// TIA Portal V20 export
FUNCTION "CallDiagnostic" : Void   // FC16, LAD
TITLE = Diagnose / Diagnostics
AUTHOR : SICAR
FAMILY : Diag
// Aufruf: Diagnose / Call of SICAR Diagnostic blocks
// stored: IsIECCheckEnabled true, SetENOAutomatically true
   VAR_TEMP
      statWStringName : WString[24];
      tempHardwareOKexample : Bool;   // REPLACE: This output can be used as an interlock for Control Modules
   END_VAR
   // Ret_Val : Ret_Val
   VAR_TEMP   // added for the SCL form of the ladder/FBD networks
      _w1 : Bool;
   END_VAR
BEGIN

REGION Network 1: Beschreibung / BLOCK INFO HEADER
   // **Betriebsart Automatik / Hand**  
   // Der Baustein ist keiner Betriebsart / Betriebsartenbereich zugeordnet.  
   // 
   // **Alarme**  
   // Der Baustein generiert keine Alarme.  
   // 
   // #### PLC-Datentypen  
   // Verwendete PLC-Datentypen für den SPS-Programmbaustein und das zugehörige WinCC-Bild.  
   // 
   // {.pageWidth}
   // ![Image](CallInterfaceSignals/de/image1.PNG)
   //  
   //  
   // #### Bausteinaufrufe 
   // Der Baustein “LSicar_InterfaceSignalsBool“ wird in diesem FB als Multi-Instanz aufgerufen, entspr. nebenstehender beispielhafter Darstellung.  
   // 
   // {.pageWidth}
   // ![Image](CallInterfaceSignals/de/image2.PNG)
   //  
   // Um einen neuen FB aufzurufen, ziehen Sie den FB in ein neues Netzwerk, wählen Sie „Multiinstanz“ aus, vergeben Sie einen Namen und parametrieren Sie den FB-Aufruf.  
   // 
   // {.pageWidth}
   // ![Image](CallInterfaceSignals/de/image3.PNG)
   //  
   //  
   // #### Weitere Hinweise 
   // 
   // #### Updateinfo 
   // 
   // #### Weitere Dokumente 
   // 
   // ![Icon](_Icon/reference.PNG)
   // 
   // ..\Library Types\LSicar_InterfaceSignalsBool.pdf
   // SIEMENS AG / (c)Copyright 2023
   // ------------------------------------------------------------------------------
   // Title:            CallDiagnostic (FC16)
   // Comment/Function: Call of SICAR Diagnostic blocks
   // Library/Family:   Diag
   // Author:           SICAR
   // Tested with:      ---
   // Engineering:      TIA Portal V19
   // Restrictions:     -
   // Requirements:     ---
   // ------------------------------------------------------------------------------
   // Change log table:
   // Version | Date | Expert in charge | Changes applied
   // -------|---------|-------------|--------------------------------------------
   // 01.00.00 | 01.01.1999 | Person x | First released version
   // 01.00.01 | 02.01.1999 | Person y | Block was Updated
END_REGION

REGION Network 2: Call: Diagnostic Profinet Devices
   // For diagnose the whole profinet devices of this PLC
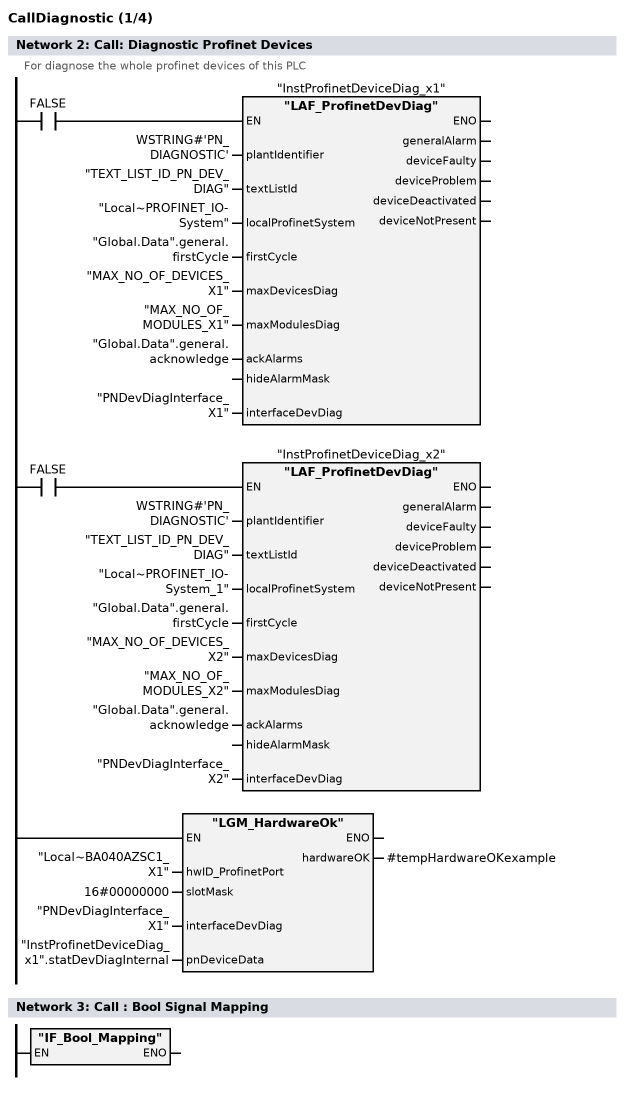
   RUNG wire#powerrail
      Contact( FALSE )
      "InstProfinetDeviceDiag_x1"(plantIdentifier := WSTRING#'PN_DIAGNOSTIC', textListId := "TEXT_LIST_ID_PN_DEV_DIAG", localProfinetSystem := "Local~PROFINET_IO-System", firstCycle := "Global.Data".general.firstCycle, maxDevicesDiag := "MAX_NO_OF_DEVICES_X1", maxModulesDiag := "MAX_NO_OF_MODULES_X1", ackAlarms := "Global.Data".general.acknowledge, hideAlarmMask :=, interfaceDevDiag := "PNDevDiagInterface_X1", generalAlarm =>, deviceFaulty =>, deviceProblem =>, deviceDeactivated =>, deviceNotPresent =>)
   END_RUNG
   RUNG wire#powerrail
      Contact( FALSE )
      "InstProfinetDeviceDiag_x2"(plantIdentifier := WSTRING#'PN_DIAGNOSTIC', textListId := "TEXT_LIST_ID_PN_DEV_DIAG", localProfinetSystem := "Local~PROFINET_IO-System_1", firstCycle := "Global.Data".general.firstCycle, maxDevicesDiag := "MAX_NO_OF_DEVICES_X2", maxModulesDiag := "MAX_NO_OF_MODULES_X2", ackAlarms := "Global.Data".general.acknowledge, hideAlarmMask :=, interfaceDevDiag := "PNDevDiagInterface_X2", generalAlarm =>, deviceFaulty =>, deviceProblem =>, deviceDeactivated =>, deviceNotPresent =>)
   END_RUNG
   RUNG wire#powerrail
      "LGM_HardwareOk"(hwID_ProfinetPort := "Local~BA040AZSC1_X1", slotMask := 16#00000000, interfaceDevDiag := "PNDevDiagInterface_X1", pnDeviceData := "InstProfinetDeviceDiag_x1".statDevDiagInternal, hardwareOK => #tempHardwareOKexample)
   END_RUNG
   // the same network as SCL:
   IF FALSE THEN
       "InstProfinetDeviceDiag_x1"(plantIdentifier := WSTRING#'PN_DIAGNOSTIC',   // "LAF_ProfinetDevDiag"
                               textListId := "TEXT_LIST_ID_PN_DEV_DIAG",
                               localProfinetSystem := "Local~PROFINET_IO-System",
                               firstCycle := "Global.Data".general.firstCycle,
                               maxDevicesDiag := "MAX_NO_OF_DEVICES_X1",
                               maxModulesDiag := "MAX_NO_OF_MODULES_X1",
                               ackAlarms := "Global.Data".general.acknowledge,
                               interfaceDevDiag := "PNDevDiagInterface_X1");
       "InstProfinetDeviceDiag_x2"(plantIdentifier := WSTRING#'PN_DIAGNOSTIC',   // "LAF_ProfinetDevDiag"
                               textListId := "TEXT_LIST_ID_PN_DEV_DIAG",
                               localProfinetSystem := "Local~PROFINET_IO-System_1",
                               firstCycle := "Global.Data".general.firstCycle,
                               maxDevicesDiag := "MAX_NO_OF_DEVICES_X2",
                               maxModulesDiag := "MAX_NO_OF_MODULES_X2",
                               ackAlarms := "Global.Data".general.acknowledge,
                               interfaceDevDiag := "PNDevDiagInterface_X2");
   END_IF;
   "LGM_HardwareOk"(hwID_ProfinetPort := "Local~BA040AZSC1_X1",
                    slotMask := 16#00000000,
                    interfaceDevDiag := "PNDevDiagInterface_X1",
                    pnDeviceData := "InstProfinetDeviceDiag_x1".statDevDiagInternal,
                    hardwareOK => #tempHardwareOKexample);
END_REGION

REGION Network 3: Call : Bool Signal Mapping
   RUNG wire#powerrail
      "IF_Bool_Mapping"()
   END_RUNG
   // the same network as SCL:
   "IF_Bool_Mapping"();
END_REGION

REGION Network 4: Call: Diagnostic Bool Interface Signals
   // Call the interface bool blocks to show boolean signals on the HMI
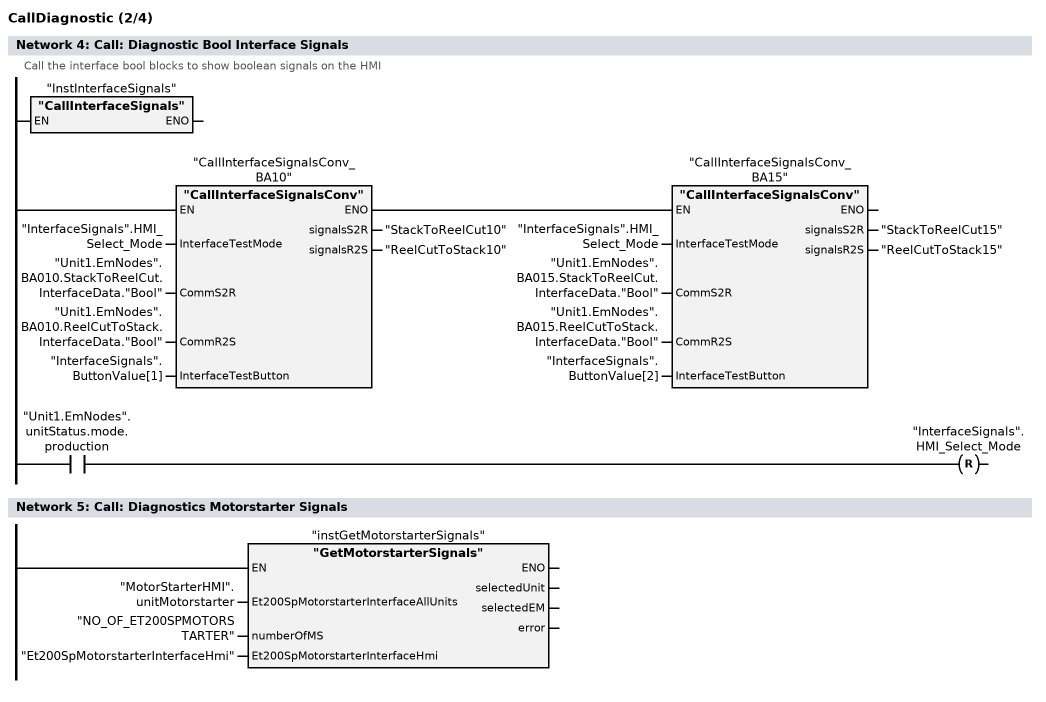
   RUNG wire#powerrail
      "InstInterfaceSignals"()
   END_RUNG
   RUNG wire#powerrail
      "CallInterfaceSignalsConv_BA10"(InterfaceTestMode := "InterfaceSignals".HMI_Select_Mode, CommS2R := "Unit1.EmNodes".BA010.StackToReelCut.InterfaceData."Bool", CommR2S := "Unit1.EmNodes".BA010.ReelCutToStack.InterfaceData."Bool", InterfaceTestButton := "InterfaceSignals".ButtonValue[1], signalsS2R => "StackToReelCut10", signalsR2S => "ReelCutToStack10")
      "CallInterfaceSignalsConv_BA15"(InterfaceTestMode := "InterfaceSignals".HMI_Select_Mode, CommS2R := "Unit1.EmNodes".BA015.StackToReelCut.InterfaceData."Bool", CommR2S := "Unit1.EmNodes".BA015.ReelCutToStack.InterfaceData."Bool", InterfaceTestButton := "InterfaceSignals".ButtonValue[2], signalsS2R => "StackToReelCut15", signalsR2S => "ReelCutToStack15")
   END_RUNG
   RUNG wire#powerrail
      Contact( "Unit1.EmNodes".unitStatus.mode.production )
      R_Coil( "InterfaceSignals".HMI_Select_Mode )
   END_RUNG
   // the same network as SCL:
   "InstInterfaceSignals"();   // "CallInterfaceSignals"
   "CallInterfaceSignalsConv_BA10"(InterfaceTestMode := "InterfaceSignals".HMI_Select_Mode,   // "CallInterfaceSignalsConv"
                           CommS2R := "Unit1.EmNodes".BA010.StackToReelCut.InterfaceData."Bool",
                           CommR2S := "Unit1.EmNodes".BA010.ReelCutToStack.InterfaceData."Bool",
                           InterfaceTestButton := "InterfaceSignals".ButtonValue[1],
                           signalsS2R => "StackToReelCut10",
                           signalsR2S => "ReelCutToStack10",
                           ENO => #_w1);
   IF #_w1 THEN
       "CallInterfaceSignalsConv_BA15"(InterfaceTestMode := "InterfaceSignals".HMI_Select_Mode,   // "CallInterfaceSignalsConv"
                               CommS2R := "Unit1.EmNodes".BA015.StackToReelCut.InterfaceData."Bool",
                               CommR2S := "Unit1.EmNodes".BA015.ReelCutToStack.InterfaceData."Bool",
                               InterfaceTestButton := "InterfaceSignals".ButtonValue[2],
                               signalsS2R => "StackToReelCut15",
                               signalsR2S => "ReelCutToStack15");
   END_IF;
   IF "Unit1.EmNodes".unitStatus.mode.production THEN "InterfaceSignals".HMI_Select_Mode := FALSE; END_IF;
END_REGION

REGION Network 5: Call: Diagnostics Motorstarter Signals
   RUNG wire#powerrail
      "instGetMotorstarterSignals"(Et200SpMotorstarterInterfaceAllUnits := "MotorStarterHMI".unitMotorstarter, numberOfMS := "NO_OF_ET200SPMOTORSTARTER", Et200SpMotorstarterInterfaceHmi := "Et200SpMotorstarterInterfaceHmi", selectedUnit =>, selectedEM =>, error =>)
   END_RUNG
   // the same network as SCL:
   "instGetMotorstarterSignals"(Et200SpMotorstarterInterfaceAllUnits := "MotorStarterHMI".unitMotorstarter,   // "GetMotorstarterSignals"
                           numberOfMS := "NO_OF_ET200SPMOTORSTARTER",
                           Et200SpMotorstarterInterfaceHmi := "Et200SpMotorstarterInterfaceHmi");
END_REGION

REGION Network 6: Call: Diagnostics Drives
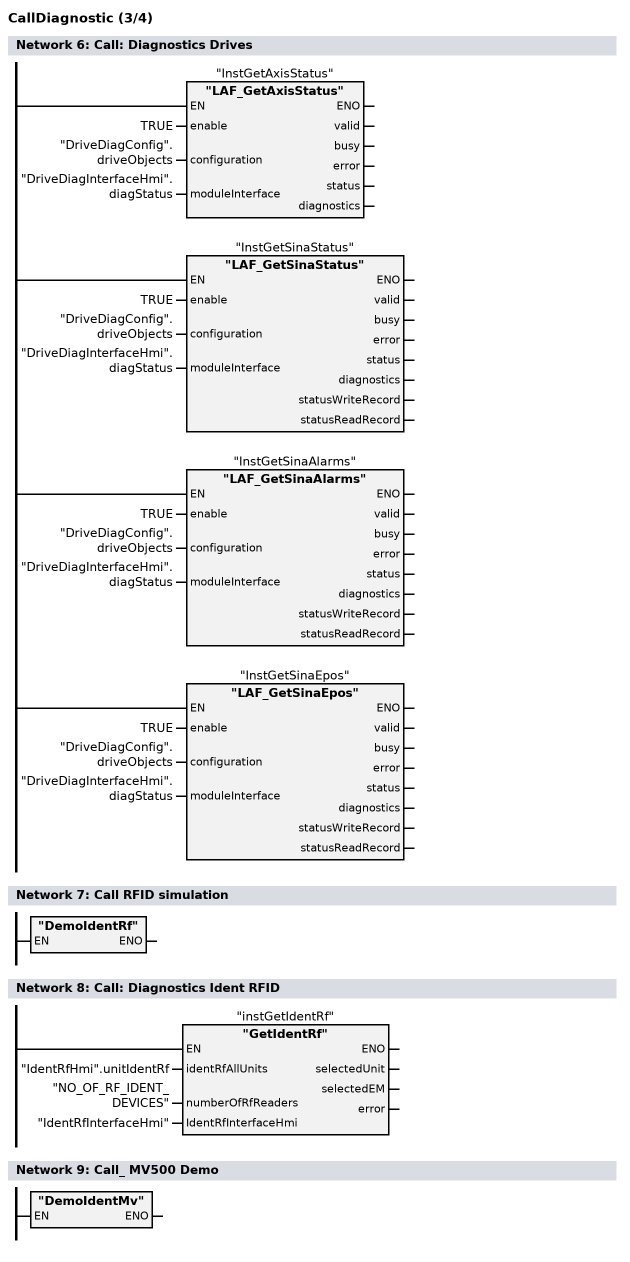
   RUNG wire#powerrail
      "InstGetAxisStatus"(enable := TRUE, configuration := "DriveDiagConfig".driveObjects, moduleInterface := "DriveDiagInterfaceHmi".diagStatus, valid =>, busy =>, error =>, status =>, diagnostics =>)
   END_RUNG
   RUNG wire#powerrail
      "InstGetSinaStatus"(enable := TRUE, configuration := "DriveDiagConfig".driveObjects, moduleInterface := "DriveDiagInterfaceHmi".diagStatus, valid =>, busy =>, error =>, status =>, diagnostics =>, statusWriteRecord =>, statusReadRecord =>)
   END_RUNG
   RUNG wire#powerrail
      "InstGetSinaAlarms"(enable := TRUE, configuration := "DriveDiagConfig".driveObjects, moduleInterface := "DriveDiagInterfaceHmi".diagStatus, valid =>, busy =>, error =>, status =>, diagnostics =>, statusWriteRecord =>, statusReadRecord =>)
   END_RUNG
   RUNG wire#powerrail
      "InstGetSinaEpos"(enable := TRUE, configuration := "DriveDiagConfig".driveObjects, moduleInterface := "DriveDiagInterfaceHmi".diagStatus, valid =>, busy =>, error =>, status =>, diagnostics =>, statusWriteRecord =>, statusReadRecord =>)
   END_RUNG
   // the same network as SCL:
   "InstGetAxisStatus"(enable := TRUE,   // "LAF_GetAxisStatus"
                       configuration := "DriveDiagConfig".driveObjects,
                       moduleInterface := "DriveDiagInterfaceHmi".diagStatus);
   "InstGetSinaStatus"(enable := TRUE,   // "LAF_GetSinaStatus"
                       configuration := "DriveDiagConfig".driveObjects,
                       moduleInterface := "DriveDiagInterfaceHmi".diagStatus);
   "InstGetSinaAlarms"(enable := TRUE,   // "LAF_GetSinaAlarms"
                       configuration := "DriveDiagConfig".driveObjects,
                       moduleInterface := "DriveDiagInterfaceHmi".diagStatus);
   "InstGetSinaEpos"(enable := TRUE,   // "LAF_GetSinaEpos"
                     configuration := "DriveDiagConfig".driveObjects,
                     moduleInterface := "DriveDiagInterfaceHmi".diagStatus);
END_REGION

REGION Network 7: Call RFID simulation
   RUNG wire#powerrail
      "DemoIdentRf"()
   END_RUNG
   // the same network as SCL:
   "DemoIdentRf"();
END_REGION

REGION Network 8: Call: Diagnostics Ident RFID
   RUNG wire#powerrail
      "instGetIdentRf"(identRfAllUnits := "IdentRfHmi".unitIdentRf, numberOfRfReaders := "NO_OF_RF_IDENT_DEVICES", IdentRfInterfaceHmi := "IdentRfInterfaceHmi", selectedUnit =>, selectedEM =>, error =>)
   END_RUNG
   // the same network as SCL:
   "instGetIdentRf"(identRfAllUnits := "IdentRfHmi".unitIdentRf,   // "GetIdentRf"
                    numberOfRfReaders := "NO_OF_RF_IDENT_DEVICES",
                    IdentRfInterfaceHmi := "IdentRfInterfaceHmi");
END_REGION

REGION Network 9: Call_ MV500 Demo
   RUNG wire#powerrail
      "DemoIdentMv"()
   END_RUNG
   // the same network as SCL:
   "DemoIdentMv"();
END_REGION

REGION Network 10: Call: Diagnosticsa Ident MV
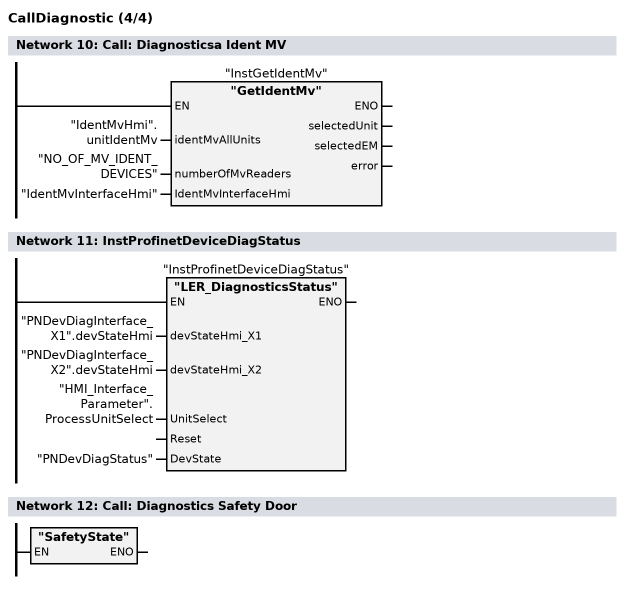
   RUNG wire#powerrail
      "InstGetIdentMv"(identMvAllUnits := "IdentMvHmi".unitIdentMv, numberOfMvReaders := "NO_OF_MV_IDENT_DEVICES", IdentMvInterfaceHmi := "IdentMvInterfaceHmi", selectedUnit =>, selectedEM =>, error =>)
   END_RUNG
   // the same network as SCL:
   "InstGetIdentMv"(identMvAllUnits := "IdentMvHmi".unitIdentMv,   // "GetIdentMv"
                    numberOfMvReaders := "NO_OF_MV_IDENT_DEVICES",
                    IdentMvInterfaceHmi := "IdentMvInterfaceHmi");
END_REGION

REGION Network 11: InstProfinetDeviceDiagStatus
   RUNG wire#powerrail
      "InstProfinetDeviceDiagStatus"(devStateHmi_X1 := "PNDevDiagInterface_X1".devStateHmi, devStateHmi_X2 := "PNDevDiagInterface_X2".devStateHmi, UnitSelect := "HMI_Interface_Parameter".ProcessUnitSelect, Reset :=, DevState := "PNDevDiagStatus")
   END_RUNG
   // the same network as SCL:
   "InstProfinetDeviceDiagStatus"(devStateHmi_X1 := "PNDevDiagInterface_X1".devStateHmi,   // "LER_DiagnosticsStatus"
                           devStateHmi_X2 := "PNDevDiagInterface_X2".devStateHmi,
                           UnitSelect := "HMI_Interface_Parameter".ProcessUnitSelect,
                           DevState := "PNDevDiagStatus");
END_REGION

REGION Network 12: Call: Diagnostics Safety Door
   RUNG wire#powerrail
      "SafetyState"()
   END_RUNG
   // the same network as SCL:
   "SafetyState"();
END_REGION
END_FUNCTION
